FUNCTION_BLOCK InstantTreeStrategyExecutor EXTENDS CNM_AbstractObject.Object IMPLEMENTS CNM_CollectionInterfaces.IInstantTreeStrategy
VAR
	tree :ITreeHelper;
END_VAR

METHOD INTERNAL assignTree
VAR_INPUT
	tree :ITreeHelper;
END_VAR
THIS^.tree := tree;
END_METHOD

(*

## Short summary

This abstract property returns the class name of the concrete object, 
which is useful for logging/debugging purpose.

.. <legal notes>

legal notes
=================
| SPDX-FileCopyrightText: © 2022 ekvip automation GmbH <info@ekvip.de>
| SPDX-License-Identifier: Apache-2.0
| For details check: Apache-2.0_

.. _Apache-2.0: https://www.apache.org/licenses/LICENSE-2.0

.. </legal notes>

*)
PROPERTY className : CNM_AbstractObject.ClassName
GET
className := 'CNM_Collections.InstantTreeStrategyExecutor';
END_GET
END_PROPERTY

(*

## Short summary

This method inserts all elements of a collection into the tree
This takes only one cycle 

.. <legal notes>

legal notes
=================
| SPDX-FileCopyrightText: © 2022 ekvip automation GmbH <info@ekvip.de>
| SPDX-License-Identifier: Apache-2.0
| For details check: Apache-2.0_

.. _Apache-2.0: https://www.apache.org/licenses/LICENSE-2.0

.. </legal notes>


**Return:** ``SingleExecutionResult.SUCCESS``: operation successful
	``SingleExecutionResult.ERROR``: out of memory
	``SingleExecutionResult.ABORTED``: collection to insert wasn't valid

*)
METHOD insertCollection : CNM_CollectionInterfaces.CNM_ReturnTypes.SingleExecutionResult
VAR_INPUT
	(*The collection that should be inserted*)
	collection	: CNM_CollectionInterfaces.ICollection;
END_VAR
insertCollection := THIS^.tree.instantInsertCollection(collection := collection);
END_METHOD

END_FUNCTION_BLOCK

(* stored: Version 1.1.0.1, ProductVersion 3.1.4026.13
   POU InstantTreeStrategyExecutor: Id {cc0f6046-cde8-4b84-8583-f52cb67fcdd1}, SpecialFunc None
   Method assignTree: Id {5882d3f5-c750-4312-838d-a43a2f5d7bd7}
   Property className: Id {1e81ccae-9288-46ba-8df4-94db5ed69ff2}
   Get Get: Id {738bb93b-eb6e-4cf6-a6c5-d5103ce4f986}
   Method insertCollection: Id {6f7f49f9-33c8-4bcb-acc8-2c0ea1c24633} *)
